// TIA Portal V20 export
TYPE "type_emRelations_em6_SoftCam"
// stored: Access Published, Namespace Unit1
   STRUCT
      finalRollerFrontAxisX : Struct
         cathode : "LER_typeSoftcamControlNodes";
         anode : "LER_typeSoftcamControlNodes";
         Pos2 { S7_SetPoint := 'True'} : "LER_typeSoftcamControlNodes";
         Pos3 { S7_SetPoint := 'True'} : "LER_typeSoftcamControlNodes";
         Pos4 { S7_SetPoint := 'True'} : "LER_typeSoftcamControlNodes";
         Pos5 { S7_SetPoint := 'True'} : "LER_typeSoftcamControlNodes";
         Pos6 { S7_SetPoint := 'True'} : "LER_typeSoftcamControlNodes";
         Pos7 { S7_SetPoint := 'True'} : "LER_typeSoftcamControlNodes";
         Pos8 { S7_SetPoint := 'True'} : "LER_typeSoftcamControlNodes";
         Pos9 { S7_SetPoint := 'True'} : "LER_typeSoftcamControlNodes";
         Pos10 { S7_SetPoint := 'True'} : "LER_typeSoftcamControlNodes";
         Pos11 { S7_SetPoint := 'True'} : "LER_typeSoftcamControlNodes";
         Pos12 { S7_SetPoint := 'True'} : "LER_typeSoftcamControlNodes";
         Pos13 { S7_SetPoint := 'True'} : "LER_typeSoftcamControlNodes";
         Pos14 { S7_SetPoint := 'True'} : "LER_typeSoftcamControlNodes";
         Pos15 { S7_SetPoint := 'True'} : "LER_typeSoftcamControlNodes";
      END_STRUCT;
      finalRollerRearAxisX : Struct
         cathode : "LER_typeSoftcamControlNodes";
         anode : "LER_typeSoftcamControlNodes";
         Pos2 { S7_SetPoint := 'True'} : "LER_typeSoftcamControlNodes";
         Pos3 { S7_SetPoint := 'True'} : "LER_typeSoftcamControlNodes";
         Pos4 { S7_SetPoint := 'True'} : "LER_typeSoftcamControlNodes";
         Pos5 { S7_SetPoint := 'True'} : "LER_typeSoftcamControlNodes";
         Pos6 { S7_SetPoint := 'True'} : "LER_typeSoftcamControlNodes";
         Pos7 { S7_SetPoint := 'True'} : "LER_typeSoftcamControlNodes";
         Pos8 { S7_SetPoint := 'True'} : "LER_typeSoftcamControlNodes";
         Pos9 { S7_SetPoint := 'True'} : "LER_typeSoftcamControlNodes";
         Pos10 { S7_SetPoint := 'True'} : "LER_typeSoftcamControlNodes";
         Pos11 { S7_SetPoint := 'True'} : "LER_typeSoftcamControlNodes";
         Pos12 { S7_SetPoint := 'True'} : "LER_typeSoftcamControlNodes";
         Pos13 { S7_SetPoint := 'True'} : "LER_typeSoftcamControlNodes";
         Pos14 { S7_SetPoint := 'True'} : "LER_typeSoftcamControlNodes";
         Pos15 { S7_SetPoint := 'True'} : "LER_typeSoftcamControlNodes";
      END_STRUCT;
      mendrelAnodeFrontAxisY : Struct
         backward : "LER_typeSoftcamControlNodes";
         forward : "LER_typeSoftcamControlNodes";
         Pos2 { S7_SetPoint := 'True'} : "LER_typeSoftcamControlNodes";
         Pos3 { S7_SetPoint := 'True'} : "LER_typeSoftcamControlNodes";
         Pos4 { S7_SetPoint := 'True'} : "LER_typeSoftcamControlNodes";
         Pos5 { S7_SetPoint := 'True'} : "LER_typeSoftcamControlNodes";
         Pos6 { S7_SetPoint := 'True'} : "LER_typeSoftcamControlNodes";
         Pos7 { S7_SetPoint := 'True'} : "LER_typeSoftcamControlNodes";
         Pos8 { S7_SetPoint := 'True'} : "LER_typeSoftcamControlNodes";
         Pos9 { S7_SetPoint := 'True'} : "LER_typeSoftcamControlNodes";
         Pos10 { S7_SetPoint := 'True'} : "LER_typeSoftcamControlNodes";
         Pos11 { S7_SetPoint := 'True'} : "LER_typeSoftcamControlNodes";
         Pos12 { S7_SetPoint := 'True'} : "LER_typeSoftcamControlNodes";
         Pos13 { S7_SetPoint := 'True'} : "LER_typeSoftcamControlNodes";
         Pos14 { S7_SetPoint := 'True'} : "LER_typeSoftcamControlNodes";
         Pos15 { S7_SetPoint := 'True'} : "LER_typeSoftcamControlNodes";
      END_STRUCT;
      mendrelAnodeFrontAxisZ : Struct
         up : "LER_typeSoftcamControlNodes";
         down : "LER_typeSoftcamControlNodes";
         Pos2 { S7_SetPoint := 'True'} : "LER_typeSoftcamControlNodes";
         Pos3 { S7_SetPoint := 'True'} : "LER_typeSoftcamControlNodes";
         Pos4 { S7_SetPoint := 'True'} : "LER_typeSoftcamControlNodes";
         Pos5 { S7_SetPoint := 'True'} : "LER_typeSoftcamControlNodes";
         Pos6 { S7_SetPoint := 'True'} : "LER_typeSoftcamControlNodes";
         Pos7 { S7_SetPoint := 'True'} : "LER_typeSoftcamControlNodes";
         Pos8 { S7_SetPoint := 'True'} : "LER_typeSoftcamControlNodes";
         Pos9 { S7_SetPoint := 'True'} : "LER_typeSoftcamControlNodes";
         Pos10 { S7_SetPoint := 'True'} : "LER_typeSoftcamControlNodes";
         Pos11 { S7_SetPoint := 'True'} : "LER_typeSoftcamControlNodes";
         Pos12 { S7_SetPoint := 'True'} : "LER_typeSoftcamControlNodes";
         Pos13 { S7_SetPoint := 'True'} : "LER_typeSoftcamControlNodes";
         Pos14 { S7_SetPoint := 'True'} : "LER_typeSoftcamControlNodes";
         Pos15 { S7_SetPoint := 'True'} : "LER_typeSoftcamControlNodes";
      END_STRUCT;
      mendrelAnodeRearAxisY : Struct
         backward : "LER_typeSoftcamControlNodes";
         forward : "LER_typeSoftcamControlNodes";
         Pos2 { S7_SetPoint := 'True'} : "LER_typeSoftcamControlNodes";
         Pos3 { S7_SetPoint := 'True'} : "LER_typeSoftcamControlNodes";
         Pos4 { S7_SetPoint := 'True'} : "LER_typeSoftcamControlNodes";
         Pos5 { S7_SetPoint := 'True'} : "LER_typeSoftcamControlNodes";
         Pos6 { S7_SetPoint := 'True'} : "LER_typeSoftcamControlNodes";
         Pos7 { S7_SetPoint := 'True'} : "LER_typeSoftcamControlNodes";
         Pos8 { S7_SetPoint := 'True'} : "LER_typeSoftcamControlNodes";
         Pos9 { S7_SetPoint := 'True'} : "LER_typeSoftcamControlNodes";
         Pos10 { S7_SetPoint := 'True'} : "LER_typeSoftcamControlNodes";
         Pos11 { S7_SetPoint := 'True'} : "LER_typeSoftcamControlNodes";
         Pos12 { S7_SetPoint := 'True'} : "LER_typeSoftcamControlNodes";
         Pos13 { S7_SetPoint := 'True'} : "LER_typeSoftcamControlNodes";
         Pos14 { S7_SetPoint := 'True'} : "LER_typeSoftcamControlNodes";
         Pos15 { S7_SetPoint := 'True'} : "LER_typeSoftcamControlNodes";
      END_STRUCT;
      mendrelAnodeRearAxisZ : Struct
         up : "LER_typeSoftcamControlNodes";
         down : "LER_typeSoftcamControlNodes";
         Pos2 { S7_SetPoint := 'True'} : "LER_typeSoftcamControlNodes";
         Pos3 { S7_SetPoint := 'True'} : "LER_typeSoftcamControlNodes";
         Pos4 { S7_SetPoint := 'True'} : "LER_typeSoftcamControlNodes";
         Pos5 { S7_SetPoint := 'True'} : "LER_typeSoftcamControlNodes";
         Pos6 { S7_SetPoint := 'True'} : "LER_typeSoftcamControlNodes";
         Pos7 { S7_SetPoint := 'True'} : "LER_typeSoftcamControlNodes";
         Pos8 { S7_SetPoint := 'True'} : "LER_typeSoftcamControlNodes";
         Pos9 { S7_SetPoint := 'True'} : "LER_typeSoftcamControlNodes";
         Pos10 { S7_SetPoint := 'True'} : "LER_typeSoftcamControlNodes";
         Pos11 { S7_SetPoint := 'True'} : "LER_typeSoftcamControlNodes";
         Pos12 { S7_SetPoint := 'True'} : "LER_typeSoftcamControlNodes";
         Pos13 { S7_SetPoint := 'True'} : "LER_typeSoftcamControlNodes";
         Pos14 { S7_SetPoint := 'True'} : "LER_typeSoftcamControlNodes";
         Pos15 { S7_SetPoint := 'True'} : "LER_typeSoftcamControlNodes";
      END_STRUCT;
      mendrelCathodeFrontAxisY : Struct
         backward : "LER_typeSoftcamControlNodes";
         forward : "LER_typeSoftcamControlNodes";
         Pos2 { S7_SetPoint := 'True'} : "LER_typeSoftcamControlNodes";
         Pos3 { S7_SetPoint := 'True'} : "LER_typeSoftcamControlNodes";
         Pos4 { S7_SetPoint := 'True'} : "LER_typeSoftcamControlNodes";
         Pos5 { S7_SetPoint := 'True'} : "LER_typeSoftcamControlNodes";
         Pos6 { S7_SetPoint := 'True'} : "LER_typeSoftcamControlNodes";
         Pos7 { S7_SetPoint := 'True'} : "LER_typeSoftcamControlNodes";
         Pos8 { S7_SetPoint := 'True'} : "LER_typeSoftcamControlNodes";
         Pos9 { S7_SetPoint := 'True'} : "LER_typeSoftcamControlNodes";
         Pos10 { S7_SetPoint := 'True'} : "LER_typeSoftcamControlNodes";
         Pos11 { S7_SetPoint := 'True'} : "LER_typeSoftcamControlNodes";
         Pos12 { S7_SetPoint := 'True'} : "LER_typeSoftcamControlNodes";
         Pos13 { S7_SetPoint := 'True'} : "LER_typeSoftcamControlNodes";
         Pos14 { S7_SetPoint := 'True'} : "LER_typeSoftcamControlNodes";
         Pos15 { S7_SetPoint := 'True'} : "LER_typeSoftcamControlNodes";
      END_STRUCT;
      mendrelCathodeFrontAxisZ : Struct
         up : "LER_typeSoftcamControlNodes";
         down : "LER_typeSoftcamControlNodes";
         Pos2 { S7_SetPoint := 'True'} : "LER_typeSoftcamControlNodes";
         Pos3 { S7_SetPoint := 'True'} : "LER_typeSoftcamControlNodes";
         Pos4 { S7_SetPoint := 'True'} : "LER_typeSoftcamControlNodes";
         Pos5 { S7_SetPoint := 'True'} : "LER_typeSoftcamControlNodes";
         Pos6 { S7_SetPoint := 'True'} : "LER_typeSoftcamControlNodes";
         Pos7 { S7_SetPoint := 'True'} : "LER_typeSoftcamControlNodes";
         Pos8 { S7_SetPoint := 'True'} : "LER_typeSoftcamControlNodes";
         Pos9 { S7_SetPoint := 'True'} : "LER_typeSoftcamControlNodes";
         Pos10 { S7_SetPoint := 'True'} : "LER_typeSoftcamControlNodes";
         Pos11 { S7_SetPoint := 'True'} : "LER_typeSoftcamControlNodes";
         Pos12 { S7_SetPoint := 'True'} : "LER_typeSoftcamControlNodes";
         Pos13 { S7_SetPoint := 'True'} : "LER_typeSoftcamControlNodes";
         Pos14 { S7_SetPoint := 'True'} : "LER_typeSoftcamControlNodes";
         Pos15 { S7_SetPoint := 'True'} : "LER_typeSoftcamControlNodes";
      END_STRUCT;
      mendrelCathodeRearAxisY : Struct
         backward : "LER_typeSoftcamControlNodes";
         forward : "LER_typeSoftcamControlNodes";
         Pos2 { S7_SetPoint := 'True'} : "LER_typeSoftcamControlNodes";
         Pos3 { S7_SetPoint := 'True'} : "LER_typeSoftcamControlNodes";
         Pos4 { S7_SetPoint := 'True'} : "LER_typeSoftcamControlNodes";
         Pos5 { S7_SetPoint := 'True'} : "LER_typeSoftcamControlNodes";
         Pos6 { S7_SetPoint := 'True'} : "LER_typeSoftcamControlNodes";
         Pos7 { S7_SetPoint := 'True'} : "LER_typeSoftcamControlNodes";
         Pos8 { S7_SetPoint := 'True'} : "LER_typeSoftcamControlNodes";
         Pos9 { S7_SetPoint := 'True'} : "LER_typeSoftcamControlNodes";
         Pos10 { S7_SetPoint := 'True'} : "LER_typeSoftcamControlNodes";
         Pos11 { S7_SetPoint := 'True'} : "LER_typeSoftcamControlNodes";
         Pos12 { S7_SetPoint := 'True'} : "LER_typeSoftcamControlNodes";
         Pos13 { S7_SetPoint := 'True'} : "LER_typeSoftcamControlNodes";
         Pos14 { S7_SetPoint := 'True'} : "LER_typeSoftcamControlNodes";
         Pos15 { S7_SetPoint := 'True'} : "LER_typeSoftcamControlNodes";
      END_STRUCT;
      mendrelCathodeRearAxisZ : Struct
         up : "LER_typeSoftcamControlNodes";
         down : "LER_typeSoftcamControlNodes";
         Pos2 { S7_SetPoint := 'True'} : "LER_typeSoftcamControlNodes";
         Pos3 { S7_SetPoint := 'True'} : "LER_typeSoftcamControlNodes";
         Pos4 { S7_SetPoint := 'True'} : "LER_typeSoftcamControlNodes";
         Pos5 { S7_SetPoint := 'True'} : "LER_typeSoftcamControlNodes";
         Pos6 { S7_SetPoint := 'True'} : "LER_typeSoftcamControlNodes";
         Pos7 { S7_SetPoint := 'True'} : "LER_typeSoftcamControlNodes";
         Pos8 { S7_SetPoint := 'True'} : "LER_typeSoftcamControlNodes";
         Pos9 { S7_SetPoint := 'True'} : "LER_typeSoftcamControlNodes";
         Pos10 { S7_SetPoint := 'True'} : "LER_typeSoftcamControlNodes";
         Pos11 { S7_SetPoint := 'True'} : "LER_typeSoftcamControlNodes";
         Pos12 { S7_SetPoint := 'True'} : "LER_typeSoftcamControlNodes";
         Pos13 { S7_SetPoint := 'True'} : "LER_typeSoftcamControlNodes";
         Pos14 { S7_SetPoint := 'True'} : "LER_typeSoftcamControlNodes";
         Pos15 { S7_SetPoint := 'True'} : "LER_typeSoftcamControlNodes";
      END_STRUCT;
      stackTableAxisZ : Struct
         wait : "LER_typeSoftcamControlNodes";
         currentJRThickness : "LER_typeSoftcamControlNodes";
         fullJRThickness : "LER_typeSoftcamControlNodes";
         Pos3 { S7_SetPoint := 'True'} : "LER_typeSoftcamControlNodes";
         Pos4 { S7_SetPoint := 'True'} : "LER_typeSoftcamControlNodes";
         Pos5 { S7_SetPoint := 'True'} : "LER_typeSoftcamControlNodes";
         Pos6 { S7_SetPoint := 'True'} : "LER_typeSoftcamControlNodes";
         Pos7 { S7_SetPoint := 'True'} : "LER_typeSoftcamControlNodes";
         Pos8 { S7_SetPoint := 'True'} : "LER_typeSoftcamControlNodes";
         Pos9 { S7_SetPoint := 'True'} : "LER_typeSoftcamControlNodes";
         Pos10 { S7_SetPoint := 'True'} : "LER_typeSoftcamControlNodes";
         Pos11 { S7_SetPoint := 'True'} : "LER_typeSoftcamControlNodes";
         Pos12 { S7_SetPoint := 'True'} : "LER_typeSoftcamControlNodes";
         Pos13 { S7_SetPoint := 'True'} : "LER_typeSoftcamControlNodes";
         Pos14 { S7_SetPoint := 'True'} : "LER_typeSoftcamControlNodes";
         Pos15 { S7_SetPoint := 'True'} : "LER_typeSoftcamControlNodes";
      END_STRUCT;
      stackTableOutFrontAxisZ : Struct
         down : "LER_typeSoftcamControlNodes";
         up : "LER_typeSoftcamControlNodes";
         Pos2 { S7_SetPoint := 'True'} : "LER_typeSoftcamControlNodes";
         Pos3 { S7_SetPoint := 'True'} : "LER_typeSoftcamControlNodes";
         Pos4 { S7_SetPoint := 'True'} : "LER_typeSoftcamControlNodes";
         Pos5 { S7_SetPoint := 'True'} : "LER_typeSoftcamControlNodes";
         Pos6 { S7_SetPoint := 'True'} : "LER_typeSoftcamControlNodes";
         Pos7 { S7_SetPoint := 'True'} : "LER_typeSoftcamControlNodes";
         Pos8 { S7_SetPoint := 'True'} : "LER_typeSoftcamControlNodes";
         Pos9 { S7_SetPoint := 'True'} : "LER_typeSoftcamControlNodes";
         Pos10 { S7_SetPoint := 'True'} : "LER_typeSoftcamControlNodes";
         Pos11 { S7_SetPoint := 'True'} : "LER_typeSoftcamControlNodes";
         Pos12 { S7_SetPoint := 'True'} : "LER_typeSoftcamControlNodes";
         Pos13 { S7_SetPoint := 'True'} : "LER_typeSoftcamControlNodes";
         Pos14 { S7_SetPoint := 'True'} : "LER_typeSoftcamControlNodes";
         Pos15 { S7_SetPoint := 'True'} : "LER_typeSoftcamControlNodes";
      END_STRUCT;
      stackTableOutRearAxisZ : Struct
         down : "LER_typeSoftcamControlNodes";
         up : "LER_typeSoftcamControlNodes";
         Pos2 { S7_SetPoint := 'True'} : "LER_typeSoftcamControlNodes";
         Pos3 { S7_SetPoint := 'True'} : "LER_typeSoftcamControlNodes";
         Pos4 { S7_SetPoint := 'True'} : "LER_typeSoftcamControlNodes";
         Pos5 { S7_SetPoint := 'True'} : "LER_typeSoftcamControlNodes";
         Pos6 { S7_SetPoint := 'True'} : "LER_typeSoftcamControlNodes";
         Pos7 { S7_SetPoint := 'True'} : "LER_typeSoftcamControlNodes";
         Pos8 { S7_SetPoint := 'True'} : "LER_typeSoftcamControlNodes";
         Pos9 { S7_SetPoint := 'True'} : "LER_typeSoftcamControlNodes";
         Pos10 { S7_SetPoint := 'True'} : "LER_typeSoftcamControlNodes";
         Pos11 { S7_SetPoint := 'True'} : "LER_typeSoftcamControlNodes";
         Pos12 { S7_SetPoint := 'True'} : "LER_typeSoftcamControlNodes";
         Pos13 { S7_SetPoint := 'True'} : "LER_typeSoftcamControlNodes";
         Pos14 { S7_SetPoint := 'True'} : "LER_typeSoftcamControlNodes";
         Pos15 { S7_SetPoint := 'True'} : "LER_typeSoftcamControlNodes";
      END_STRUCT;
   END_STRUCT;
END_TYPE
